TYPE DUT_SEW_FU_Steuern :
STRUCT

	vor					:BOOL;
	zur					:BOOL;
	speed				:REAL;
	
END_STRUCT
END_TYPE

(* stored: Version 1.1.0.1
   DUT DUT_SEW_FU_Steuern: Id {ce1e012d-31b2-4784-ae9e-577b81cee945} *)
